{attribute addProperty BoxType "EL3692-0000-0017"}
{attribute addProperty Id "SettingsAT %I*Settings_7AA6B313162"}
{attribute addProperty CRC "3751299124"}
{attribute addProperty SizeInBites "16"}
{attribute addProperty SizeInBytes "2"}
TYPE SAI_Range_Channel_DF984834 :
STRUCT
	{attribute addProperty Name "Settings"}
	Settings AT %I* : Settings_7AA6B313;
END_STRUCT
END_TYPE

(* stored: Version 1.2.0.0, ProductVersion 3.1.4024.9
   DUT SAI_Range_Channel_DF984834: Id {e5f405ac-0371-4ec6-a67a-83f00acacf4b} *)
